Omron Sysmac Studio project LS and TCP ONLY (Sysmac Studio 1.43.0.64009, StandardProject)

# Controller new_Controller_0: NX1P2-9024DT version 1.42
Task PrimaryTask (priority 4, period or condition 2000): Program0
Library OEN_Communication_V1_0_22 1.0.22 (contents left out)
Library MTCP_Server_NJNX 2.5.1 (contents left out)

VAR_GLOBAL
    D0 : BOOL;  (* at BuiltInIO://cpu/#0/Input_Bit_00 *)
    O1 : BOOL;  (* at BuiltInIO://cpu/#0/Output_Bit_00 *)
    testVar : WORD;
END_VAR

PROGRAM Program0
VAR
    FB_ModbusTCPServer : OEN\Modbus\ModbusTCP_Server;
    ModbusCoils : ARRAY[1..16] OF BOOL;
    ModbusInputs : ARRAY[1..10] OF BOOL;
    ModbusInputsRegs : ARRAY[1..10] OF WORD;
    ModbusHolding : ARRAY[1..10] OF WORD;
    ModbusAccessList : ARRAY[0..0] OF OEN\Modbus\sModbusAccess;
    testVar : WORD;
    FB_ModbusTCPClient : OEN\Modbus\ModbusTCP_Client;
    RequestTable : ARRAY[1..2] OF OEN\Modbus\sModbusReq := [(Enable := True, NodeAdr := 0, FunctionCode := Fn01_ReadCoils, Read := (StartAddressRemote := 1, StartAddressLocal := 1, Count := 3), Write := (StartAddressRemote := 0, StartAddressLocal := 0, Count := 0)), (Enable := True, NodeAdr := 0, FunctionCode := Fn01_ReadCoils, Read := (StartAddressRemote := 0, StartAddressLocal := 0, Count := 0), Write := (StartAddressRemote := 4, StartAddressLocal := 4, Count := 1))];
    ModbusCoils_Client : ARRAY[1..16] OF BOOL;
    ModbusInputs_Client : ARRAY[1..16] OF BOOL;
    ModbusInputRegs_Client : ARRAY[1..16] OF WORD;
    ModbusHolding_Client : ARRAY[1..16] OF WORD;
END_VAR
VAR_EXTERNAL
    O1 : BOOL;
    D0 : BOOL;
END_VAR

(* Section Section0: ladder, written here as Structured Text *)

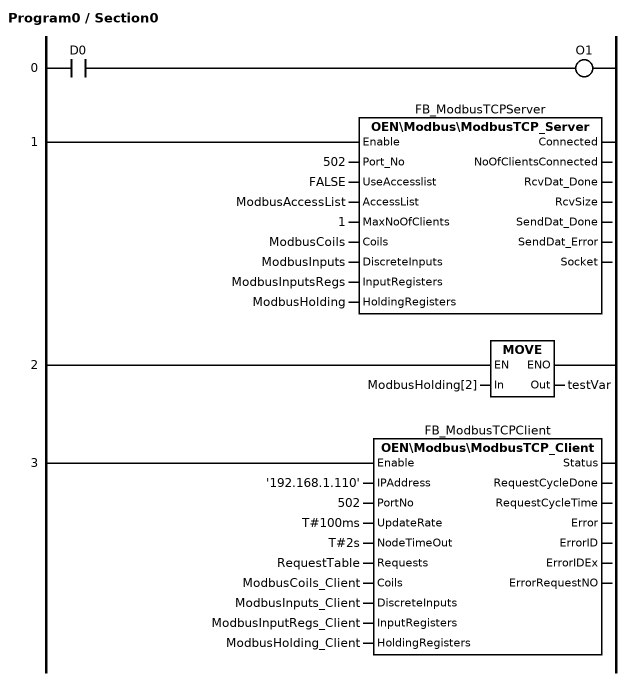
(* Rung 0 *)
O1 := D0;
(* Rung 1 *)
FB_ModbusTCPServer(Enable := TRUE, Port_No := 502, UseAccesslist := FALSE, AccessList := ModbusAccessList, MaxNoOfClients := 1, Coils := ModbusCoils, DiscreteInputs := ModbusInputs, InputRegisters := ModbusInputsRegs, HoldingRegisters := ModbusHolding);
(* Rung 2 *)
testVar := ModbusHolding[2];
(* Rung 3 *)
FB_ModbusTCPClient(Enable := TRUE, IPAddress := '192.168.1.110', PortNo := 502, UpdateRate := T#100ms, NodeTimeOut := T#2s, Requests := RequestTable, Coils := ModbusCoils_Client, DiscreteInputs := ModbusInputs_Client, InputRegisters := ModbusInputRegs_Client, HoldingRegisters := ModbusHolding_Client);
END_PROGRAM